% RSLogix 500 project P9_KOBIERSKI_M.RSS, saved by version 8.30.00.16 %
PROJECT "UNTITLED"    % processor: Bul.1763 MicroLogix 1100 Series B %

PROGRAM FILES
  LAD 2 "MAIN"  12 rungs

DATA FILES
  O0 OUTPUT  4 elements
  I1 INPUT  6 elements
  S2 STATUS  66 elements
  B3 BINARY  1 elements
  T4 TIMER  3 elements
  C5 COUNTER  1 elements
  R6 CONTROL  1 elements
  N7 INTEGER  4 elements
  F8 FLOAT  1 elements
  ST9 STRINGS  5 elements

LADDER 2 "MAIN"
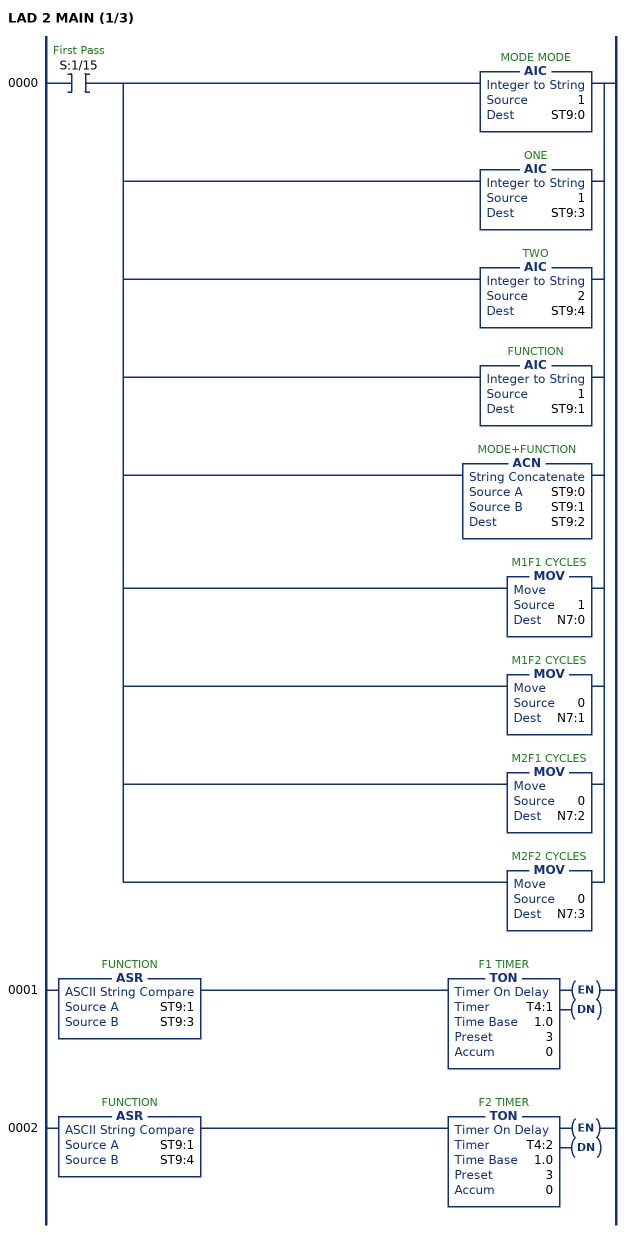
% Rung: 0 %  % edit flag set %
SOR XIC S:1/15 BST AIC 1 ST9:0 NXB AIC 1 ST9:3 NXB AIC 2 ST9:4 NXB AIC 1 ST9:1 NXB ACN ST9:0 ST9:1 ST9:2 NXB MOV 1 N7:0 NXB MOV 0 N7:1 NXB MOV 0 N7:2 NXB MOV 0 N7:3 BND EOR
%   S:1/15  "First Pass" %
%   ST9:0  MODE  "MODE" %
%   ST9:3  "ONE" %
%   ST9:4  "TWO" %
%   ST9:1  "FUNCTION" %
%   ST9:2  "MODE+FUNCTION" %
%   N7:0  "M1F1 CYCLES" %
%   N7:1  "M1F2 CYCLES" %
%   N7:2  "M2F1 CYCLES" %
%   N7:3  "M2F2 CYCLES" %
% Rung: 1 %
SOR ASR ST9:1 ST9:3 TON T4:1 1.0 3 0 EOR
%   ST9:1  "FUNCTION" %
%   ST9:3  "ONE" %
%   T4:1  "F1 TIMER" %
% Rung: 2 %
SOR ASR ST9:1 ST9:4 TON T4:2 1.0 3 0 EOR
%   ST9:1  "FUNCTION" %
%   ST9:4  "TWO" %
%   T4:2  "F2 TIMER" %

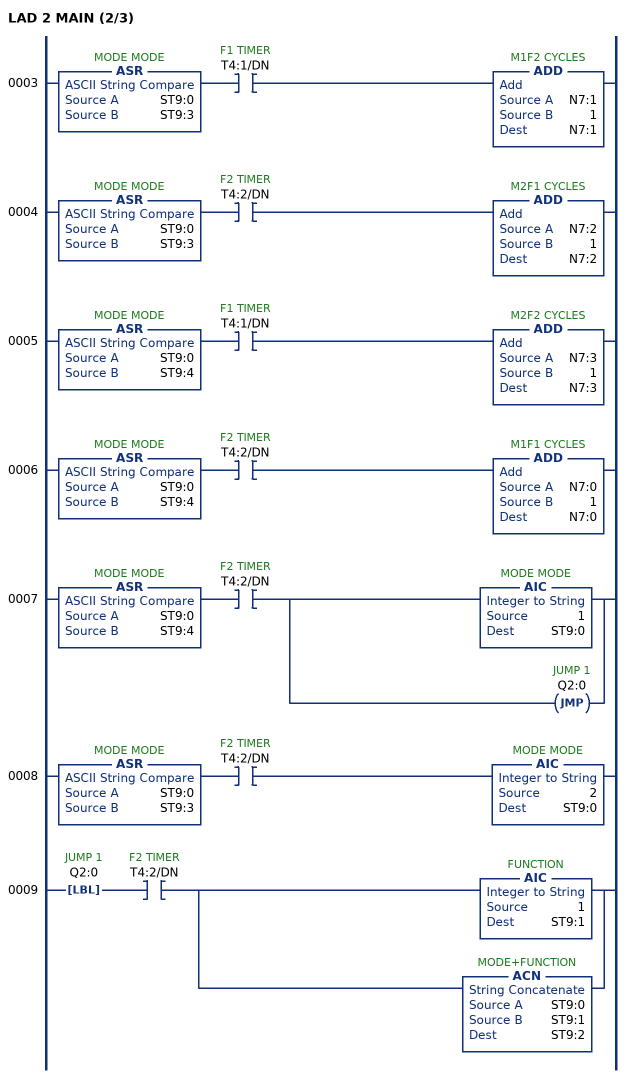
% Rung: 3 %
SOR ASR ST9:0 ST9:3 XIC T4:1/DN ADD N7:1 1 N7:1 EOR
%   ST9:0  MODE  "MODE" %
%   ST9:3  "ONE" %
%   T4:1  "F1 TIMER" %
%   N7:1  "M1F2 CYCLES" %
% Rung: 4 %
SOR ASR ST9:0 ST9:3 XIC T4:2/DN ADD N7:2 1 N7:2 EOR
%   ST9:0  MODE  "MODE" %
%   ST9:3  "ONE" %
%   T4:2  "F2 TIMER" %
%   N7:2  "M2F1 CYCLES" %
% Rung: 5 %
SOR ASR ST9:0 ST9:4 XIC T4:1/DN ADD N7:3 1 N7:3 EOR
%   ST9:0  MODE  "MODE" %
%   ST9:4  "TWO" %
%   T4:1  "F1 TIMER" %
%   N7:3  "M2F2 CYCLES" %
% Rung: 6 %
SOR ASR ST9:0 ST9:4 XIC T4:2/DN ADD N7:0 1 N7:0 EOR
%   ST9:0  MODE  "MODE" %
%   ST9:4  "TWO" %
%   T4:2  "F2 TIMER" %
%   N7:0  "M1F1 CYCLES" %
% Rung: 7 %
SOR ASR ST9:0 ST9:4 XIC T4:2/DN BST AIC 1 ST9:0 NXB JMP Q2:0 BND EOR
%   ST9:0  MODE  "MODE" %
%   ST9:4  "TWO" %
%   T4:2  "F2 TIMER" %
%   Q2:0  "JUMP 1" %
% Rung: 8 %
SOR ASR ST9:0 ST9:3 XIC T4:2/DN AIC 2 ST9:0 EOR
%   ST9:0  MODE  "MODE" %
%   ST9:3  "ONE" %
%   T4:2  "F2 TIMER" %
% Rung: 9 %
SOR LBL Q2:0 XIC T4:2/DN BST AIC 1 ST9:1 NXB ACN ST9:0 ST9:1 ST9:2 BND EOR
%   Q2:0  "JUMP 1" %
%   T4:2  "F2 TIMER" %
%   ST9:1  "FUNCTION" %
%   ST9:0  MODE  "MODE" %
%   ST9:2  "MODE+FUNCTION" %

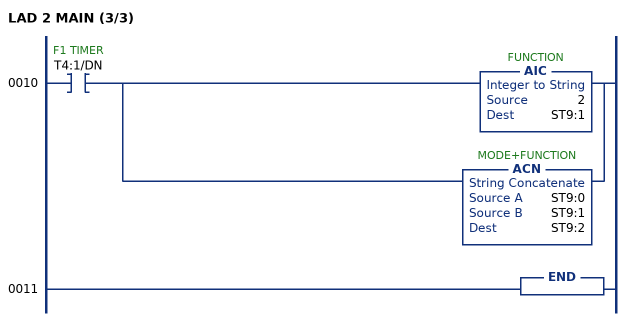
% Rung: 10 %
SOR XIC T4:1/DN BST AIC 2 ST9:1 NXB ACN ST9:0 ST9:1 ST9:2 BND EOR
%   T4:1  "F1 TIMER" %
%   ST9:1  "FUNCTION" %
%   ST9:0  MODE  "MODE" %
%   ST9:2  "MODE+FUNCTION" %
% Rung: 11 %
SOR END EOR

OTHER DOCUMENTED ADDRESSES
  B3:0/0  "START BIT"

DATA TABLE (non-zero values as saved)
DATA T4
% .PRE .ACC %
% T4:1 % 3 0
% T4:2 % 3 0
